// TIA Portal V20 export
TYPE "zm_LOGSOperationData1"
// stored: Access Published
   STRUCT
      ReadyForOperation : Bool;
      MachineInOperation : Bool;
      PartOn : Bool;
      PartReady : Bool;
   END_STRUCT;
END_TYPE
